TYPE ST_VCC :
STRUCT

(* Inputs *)
	xOPN_SW	: BOOL;
	xOvrdOpn	:	BOOL;
	xOPN_OK	: BOOL;

(* Outputs *)
	xOPN_DO	: BOOL;

END_STRUCT
END_TYPE

(* stored: Version 1.1.0.1, ProductVersion 3.1.0.24
   DUT ST_VCC: Id {f8163ff7-c34c-4425-9a0d-608ae9423340} *)
